               //start purging
               //-------------
               IF "APC".AUTOMATIC THEN 
                   IF ("APC".TI[0] <= REAL_TO_INT("PAR_MAIN".PD_PRG_TME)) AND NOT "PDI".FCH_APS  THEN 
                       //purging through V5
                       //------------------
                       IF (REAL_TO_INT("PAR_MAIN".PD_PRG_INLET_V5) = 1)   THEN 
                           "DC".V4_OP            :=  FALSE;
                           "DC".V5_OP            :=  TRUE;
                           "AC".SET_GAS_2_FLW    :=  "PAR_MAIN".PD_PRG_GAS_FLW;
                       //purging through V4
                       //------------------
                       ELSE
                           "DC".V4_OP            :=  TRUE;
                           "DC".V5_OP            :=  FALSE;
                           "AC".SET_GAS_2_FLW    :=  0.0;
                       END_IF;
                   //purging over
                   //------------
                   ELSE 
                       "DC".V4_OP            :=  FALSE;
                       "DC".V5_OP            :=  FALSE;
                       "AC".SET_GAS_2_FLW    :=  0.0;

                       #end_of_step[0] := true;                            

                   END_IF;
               END_IF;

               //calculate step time countdown
               //-----------------------------            
               "APC".ACT_TME_STE   := REAL_TO_INT("PAR_MAIN".PD_PRG_TME) - "APC".TI[0];

               #next_step[0] := 180;   

   //-step-180---level--0-------------------------------------------------------------                                                 
   //            PD: check if additional purge cycle is requested
   //---------------------------------------------------------------------------------                                                 
           180 :                                                     
               IF #next_step[0] = #active_step[0] THEN
                   "APC".OP_MSG  := "OP_MSG".BLANK;       
                   "APC".TI[0]   :=  0;            
                   #prg_cyc_cnt :=  #prg_cyc_cnt + 1;    //count amount of purge cycles                              
               END_IF;

               //delay switching to next step
               //----------------------------
               IF ("APC".TI[0] > 2) THEN
                   #end_of_step[0] := true;                            
               END_IF;

               //select next step
               //----------------
               IF (#prg_cyc_cnt >= REAL_TO_INT("PAR_MAIN".PD_AMT_PRG_CYC)) THEN
                   #next_step[0] := 200; 
               ELSE
                   #next_step[0] := 140; 
               END_IF;

   //-step-200---level--0-------------------------------------------------------------                                                 
   //            PD: pump down to 10 mbar
   //---------------------------------------------------------------------------------                                                 
           200 :                                                     
               IF #next_step[0] = #active_step[0] THEN                       
                   //reset initial temperature and power setpoints
                   //---------------------------------------------
                   "DIS".HTR_1_TMP_SET_PHA_STR   :=  0.0;
                   "DIS".HTR_2_PWR_SET_PHA_STR   :=  0.0;
                   "APC".TI[0]                   :=  0;                              // start pd time                              
                   "APC".OP_MSG                  :=  "OP_MSG".PD_10MBAR;
                   "APC".ACT_TME_STE             :=  0;
               END_IF;

               // calculate all setpoints 
               // -----------------------
               "AM_PAR_FNC_PD" (act_x_value := 0.0);

               //open vacuum valves
               //------------------
               "DC".P1_ON             := TRUE;   // main pump on
               "AC".SET_CTL_VALVE_POS := 100.0;  

               //monitor pump down time 
               //----------------------
               IF "APC".AUTOMATIC THEN 
                   IF "BM_VAC_DB".V2_ONDELAY_OVER THEN                                 // vacuum valve release
                       IF (INT_TO_REAL("APC".TI[0]) > "PAR_MAIN".PD_10_MBAR_TME) THEN    // pump down time limit exceeded?
                           "FLT".PD_TIME_10MBAR  := TRUE;
                           "APC".OP_MSG          := "OP_MSG".PD_CHECK_TIME;
                           #cont_enable[0]      := true;
                       END_IF;

                       //check end condition
                       //-------------------
                       IF ("AV".ACT_PRS_FCH < 10.0)  THEN         // p < 10 mbar ?
                           #end_of_step[0] := true;
                       END_IF; 

                   ELSE
                       "APC".TI[0]:= 0;      //keep timer on zero until vacuum valve release 
                   END_IF;
               ELSE
                   "APC".TI[0]:= 0;      //keep timer on zero until vacuum valve release 
               END_IF;

               #next_step[0] := 300; 

   //-step-300---level--0-------------------------------------------------------------                                                 
   //            PD: pump down to 1 mbar
   //---------------------------------------------------------------------------------                                                 
           300 :                                                  
               IF #next_step[0] = #active_step[0] THEN                       
                   "FLT".PD_TIME_10MBAR := FALSE;
                   "APC".OP_MSG := "OP_MSG".PD_1MBAR;
               END_IF;

               // calculate all setpoints 
               // -----------------------
               "AM_PAR_FNC_PD" (act_x_value := 0.0);

               IF (INT_TO_REAL("APC".TI[0]) > "PAR_MAIN".PD_1_MBAR_TME) THEN     // limit reached ?
                   "FLT".PD_TIME_1MBAR := TRUE;
                   "APC".OP_MSG := "OP_MSG".PD_CHECK_TIME;
                   #cont_enable[0] := true;
               END_IF;

               IF ("AV".ACT_PRS_FCH < 1.0) THEN                       // p < 1 mbar ?
                   #end_of_step[0] := true;                            
               END_IF;

               #next_step[0] := 400; 

   //-step-400---level--0-------------------------------------------------------------                                                 
   //            PD: pump down to 0.1 mbar
   //---------------------------------------------------------------------------------                                                 
           400 :                                                  
               IF #next_step[0] = #active_step[0] THEN
                   "FLT".PD_TIME_1MBAR := FALSE;
                   "APC".OP_MSG := "OP_MSG".PD_01MBAR;
               END_IF;

               // calculate all setpoints 
               // -----------------------
               "AM_PAR_FNC_PD" (act_x_value := 0.0);

               IF ( INT_TO_REAL("APC".TI[0]) > "PAR_MAIN".PD_01_MBAR_TME) THEN    // limit reached ?
                   "FLT".PD_TIME_01MBAR  := TRUE;
                   "APC".OP_MSG          := "OP_MSG".PD_CHECK_TIME;
                   #cont_enable[0]      := true;
               END_IF;

               IF ("AV".ACT_PRS_FCH < 0.1) THEN                       // p < 0.1 mbar ? 
                   #end_of_step[0] := true;                            
               END_IF;

               #next_step[0] := 500; 

   //-step-500---level--0-------------------------------------------------------------                                                 
   //            PD: pump down to 0.05 mbar
   //---------------------------------------------------------------------------------                                                 
           500 :                                                  
               IF #next_step[0] = #active_step[0] THEN
                   "FLT".PD_TIME_01MBAR := FALSE;
                   "APC".OP_MSG := "OP_MSG".PD_005MBAR;
               END_IF;

               // calculate all setpoints 
               // -----------------------
               "AM_PAR_FNC_PD" (act_x_value := 0.0);

               IF (INT_TO_REAL("APC".TI[0]) > "PAR_MAIN".PD_005_MBAR_TME) THEN   // limit reached ?
                   "FLT".PD_TIME_005MBAR := TRUE;
                   "APC".OP_MSG          := "OP_MSG".PD_CHECK_TIME;
                   #cont_enable[0]      := true;
               END_IF;

               IF ("AV".ACT_PRS_FCH < 0.05) THEN                      // p < 0.05 mbar ? 
                   #end_of_step[0] := true;                            
               END_IF;

               #next_step[0] := 600; 


   //-step-600---level--0-------------------------------------------------------------                                                 
   //            PD: pump down to final pressure
   //---------------------------------------------------------------------------------                                                 
           600 :                                                  
               IF #next_step[0] = #active_step[0] THEN
                   "FLT".PD_TIME_005MBAR := FALSE;
                   "APC".OP_MSG := "OP_MSG".PD_FINAL;
               END_IF;

               // calculate all setpoints 
               // -----------------------
               "AM_PAR_FNC_PD" (act_x_value := 0.0);

               //bypass filter activated
               //-----------------------
               IF (("CNF".ACT_DVC_CNF AND 2#1000_0000_0000_0000_0000_0000_0000_0000) = 2#1000_0000_0000_0000_0000_0000_0000_0000) THEN 

                   //close valve V3.4 to bypass filter when pressure below 5 mbar
                   //-----------------------------------------------------------
                   IF ("DIS".ACT_PRS_BYP_FIL < 5.0) THEN
                       "DC".V3_4_OP  := FALSE;
                   END_IF;

                   //set global release bit of V1.1
                   //------------------------------
                   IF NOT "PDO".V3_4 THEN
                       "DC".V1_1_REL := TRUE;
                   END_IF;

                   //check end condition
                   //-------------------
                   IF (("AV".ACT_PRS_FCH < "PAR_MAIN".PD_FINAL_PRS) AND "DC".V1_1_REL) THEN         // final presssure ?      
                       #end_of_step[0] := true;                            
                   END_IF;
               //no bypass filter
               //----------------
               ELSE
                   //check end condition
                   //-------------------
                   IF ("AV".ACT_PRS_FCH < "PAR_MAIN".PD_FINAL_PRS) THEN         // final presssure ?      
                       #end_of_step[0] := true;                            
                   END_IF;
               END_IF;

               #next_step[0] := 650; 

   //-step-650---level--0-------------------------------------------------------------                                                 
   //            PD: wait time after reaching final pressure before leak test
   //---------------------------------------------------------------------------------                                                 
           650 :                                                  
               IF #next_step[0] = #active_step[0] THEN
                   "APC".OP_MSG  := "OP_MSG".PD_WAIT_TME;
                   "APC".TI[0]   := 0;
               END_IF;

               // calculate all setpoints 
               // -----------------------
               "AM_PAR_FNC_PD" (act_x_value := 0.0);

               //remaining wait time
               //-------------------
               "APC".ACT_TME_STE   := REAL_TO_INT("PAR_MAIN".PD_WAIT_TME_FIN_PRS) - "APC".TI[0];

               //check end condition
               //-------------------
               IF ("APC".TI[0] >= (REAL_TO_INT("PAR_MAIN".PD_WAIT_TME_FIN_PRS))) THEN      
                   #end_of_step[0] := true;                            
               END_IF;

               #next_step[0] := 700; 

   //-step-700---level--0-------------------------------------------------------------                                                 
   //            PD: close vacuum valve
   //---------------------------------------------------------------------------------                                                 
           700 :                                                  
               IF #next_step[0] = #active_step[0] THEN                       
                   "APC".OP_MSG := "OP_MSG".PD_LEAK_TEST;
               END_IF;

               // calculate all setpoints 
               // -----------------------
               "AM_PAR_FNC_PD" (act_x_value := 0.0);

               "AC".SET_CTL_VALVE_POS := 0.0;                // close throttle valve
               "DC".V1_OPEN_REQ      := FALSE;               // only EKZ 2700
               "DC".V1_CLOSE_REQ     := TRUE;
               "DC".P3_ON            := FALSE;               // P3 off

               // check end condition
               //--------------------
               IF NOT "LT".V1_OPEN THEN  // closed ? 
                   #end_of_step[0] := true;                            
               END_IF;

               #next_step[0] := 800; 


   //-step-800---level--0-------------------------------------------------------------                                                 
   //            PD: do leak test
   //---------------------------------------------------------------------------------                                                 
           800 :                                                  
               IF #next_step[0] = #active_step[0] THEN                       
                   "APC".TI[0] := 0;                              // start time for leak test                              
                   #prs_leak_test_start := "AV".ACT_PRS_FCH;           // save start pressure  
               END_IF;

               //store pressure value before leak test is starting (CDP)
               //-------------------------------------------------------
               "DIS".ACT_FNC_PRS_BEF_LKT :=  #prs_leak_test_start;

               // calculate all setpoints 
               // -----------------------
               "AM_PAR_FNC_PD" (act_x_value := 0.0);

               // leakrate = (p2-p1)*V/t
               // ----------------------
               IF ("APC".TI[0] > 0) THEN 
                   //leak rate calculation with main and bypass filter
                   //-------------------------------------------------
                   IF (("CNF".ACT_DVC_CNF AND 2#1000_0000_0000_0000_0000_0000_0000_0000) = 2#1000_0000_0000_0000_0000_0000_0000_0000) THEN 
                       "AV".LRT_EKZ := ("AV".ACT_PRS_FCH - #prs_leak_test_start) * ("CNF".VOLUME_LEAK_TEST + "CNF".VOLUME_MAIN_FIL + "CNF".VOLUME_BYP_FIL) / INT_TO_REAL("APC".TI[0]);
                   //leak rate calculation only with main filter
                   //-------------------------------------------
                   ELSE
                       "AV".LRT_EKZ := ("AV".ACT_PRS_FCH - #prs_leak_test_start) * ("CNF".VOLUME_LEAK_TEST + "CNF".VOLUME_MAIN_FIL) / INT_TO_REAL("APC".TI[0]);
                   END_IF;
               END_IF;

               IF ("AV".LRT_EKZ < 0.0) THEN
                   "AV".LRT_EKZ := 0.0;
               END_IF;

               // show actual values
               // ------------------
               "DIS".ACT_LEAKR_FNC := "AV".LRT_EKZ;
               "APC".ACT_TME_STE   := REAL_TO_INT("PAR_MAIN".PD_LEAKTEST_TME) - "APC".TI[0];

               // check if leak test time is over
               //--------------------------------
               IF ("APC".TI[0] >= "PAR_MAIN".PD_LEAKTEST_TME) THEN   // time for leak test ? 
                   #end_of_step[0] := true;
               END_IF;
               #next_step[0] := 900; 


   //-step-900---level--0-------------------------------------------------------------                                                 
   //            PD: check for max. leak rate
   //---------------------------------------------------------------------------------                                                 
           900 :
               // calculate all setpoints 
               // -----------------------
               "AM_PAR_FNC_PD" (act_x_value := 0.0);

               IF ("AV".LRT_EKZ > "PAR_MAIN".PD_MAX_LEAKRATE) THEN   // max. leakrate ?                   
                   "FLT".PD_LEAKTEST := TRUE;
                   "APC".OP_MSG      := "OP_MSG".PD_CHECK_LEAK_RATE;

                   #cont_enable[0]  := true;                      // wait for continue
                   #next_step[0]    := 950; 
                   //repeat leak test
                   //----------------
                   IF "KYD".PD_NEW_LKT   THEN
                       #end_of_step[0] := true;     // next step  
                       #next_step[0] := 200;            //repeat leak test

                   END_IF;

               ELSE
                   "FLT".PD_LEAKTEST := FALSE;
                   #end_of_step[0]  := true;                      // next step                            
                   #next_step[0]    := 950; 

               END_IF;

   //-step-950--level--0-------------------------------------------------------------                                                 
   //            PD: switch vacuum pump on if next phase is melting
   //---------------------------------------------------------------------------------    

           950 :             
               IF #next_step[0] = #active_step[0] THEN                       
                   "APC".TI[0]   := 0;                           // start wait time pump  
                   "APC".OP_MSG  := "OP_MSG".BLANK;                                          
               END_IF;

               IF ("APC".PD_WITH_ME) THEN                        // with melting ?
                   "DC".P1_ON := TRUE;
                   IF "BM_VAC_DB".V2_ONDELAY_OVER THEN           // wait until V2 delay is over
                       #end_of_step[0] := true;
                   END_IF;
               ELSE                                              
                   #end_of_step[0] := true;                     // switch to next step
               END_IF;

               #next_step[0] := 1000;



   //-step-1000--level--0-------------------------------------------------------------                                                 
   //            PD: start melting or switch to idle
   //---------------------------------------------------------------------------------                                                 
           1000 :                                                  

               "APC".ACT_TME_STE := 0;
               "FLT".PD_LEAKTEST := FALSE;

               IF ("APC".PD_WITH_ME) THEN                         // with melting ?
                   "DC".MOD_ME := TRUE;                           // switch to melting
               ELSE;
                  //DC.P1_ON := FALSE;                           // stop main pump 

                   // stop drives and reset setpoint values after leaktest with drives active
                   // -----------------------------------------------------------------------
                   IF "CNF".CONF_DRV_WHILE_LRT = TRUE THEN
                       "DC".XT_LFT_UP    := FALSE;                    // stop crystal lift
                       "DC".XT_LFT_DN    := FALSE;
                       "DC".XT_LFT_FST   := FALSE;
                       "DC".XT_ROT_CW    := FALSE;                    // stop crystal rotation
                       "DC".XT_ROT_CCW   := FALSE;

                       "DC".CR_LFT_UP    := FALSE;                    // stop crucible lift
                       "DC".CR_LFT_DN    := FALSE;
                       "DC".CR_LFT_FST   := FALSE;
                       "DC".CR_ROT_CW    := FALSE;                    // stop crucible rotation
                       "DC".CR_ROT_CCW   := FALSE;

                       "AC".SET_XT_SPD := 0.0;
                       "AC".SET_XT_ROT := 0.0;
                       "AC".SET_CR_SPD := 0.0;
                       "AC".SET_CR_ROT := 0.0;
                   END_IF;

                   "DC".MOD_ID := TRUE;                           // switch to idle 
               END_IF;

               #next_step[0] := 1000;                            // E N D

   //---------------------------------------------------------------------------------                                                 
   //---------------------------------------------------------------------------------                                                 

   //-error------level--0---------------------------------------------------(error in level 0)-------------
       ELSE:                                                        
           //error code                                                //do error code
           ;        
   //------------------------------------------------------------------------------------------------------
       END_CASE;

       #start_previous := #start;                                    //save start input for next call 
       #cont_previous := "APC".CONT;                                  //save cont input for next call 
       #resume_previous := "APC".RESUME;                              //save resume input for next call
       #jump_previous := "APC".JUMP;                                  //save jump input for next call
       #single_previous := "APC".SINGLE;                              //save single input for next call
END_FUNCTION_BLOCK

FUNCTION_BLOCK "AM_ME"   // FB197, SCL
{ S7_Optimized_Access := 'FALSE' }
VERSION : 0.0
// --------------------------------------------------------------------------------
//     program     :    AM_ME
//     description :    apc melting module  
//     name        :    D. Bruess
//     date        :    04.11.99
// 
//     revision    :    change default rotation direction: xtal= ccw and cruc= cw
//     name        :    G. Eibelsh鋟ser
//     date        :    26.04.00
//     
//                     (c)CGS
//     --------------------------------------------------------------------------------
   VAR_INPUT
      start : Bool;   // start sequence, activate step 10 (impulse triggered)
   END_VAR
   VAR
      start_previous : Bool;   // start input value of last call
      cont_previous : Bool;   // cont input value of last call
      resume_previous : Bool;   // resume input value of last call
      jump_previous : Bool;   // jump input value of last call
      single_previous : Bool;   // single input value of last call
      active_step : Array[0..7] of Int;   // active step number for sequence level 0..7
      next_step : Array[0..7] of Int;   // next step number for sequence level 0..7
      hold_step : Array[0..7] of Int;   // step number of step on hold
      end_of_step : Array[0..7] of Bool;   // active step is done flag for sequence 0..7
      EndOfStep : Bool;   // default value for active step is done flag
      cont_enable : Array[0..7] of Bool;   // enable continue function
      ContEnable : Bool;   // default value for enable continue function
      cam_active : Bool;   // camera used for this step
      cruc_in_pos : Bool;   // crucible in new position
      next_step_fdr : Bool;
      check_mlt_lvl_done : Bool;
      step_switch_done : Bool;
      next_melt_step : Bool;
      act_step_fdr : Int;
      par_line : Int;   // act. line from parameter table
      par_step : Int;   // number of this step
      par_time : Int;   // time parameter for this step
      set_cr_pos_old : Real;   // old setpoint for crucible position
      htr_1_pwr_act_step : Real;
      htr_1_pwr_next_step : Real;
   END_VAR
   VAR CONSTANT
      max_amt_of_steps : Int := 21;   // maximum amount of step lines
   END_VAR
BEGIN

       "APC".STATUS := "APC".MELTING;                                  // set apc status               

       "AM_SEQUENCE_CTL" (start_p            := #start,               // control sequence
                        start_previous_p   := #start_previous,
                        cont_previous_p    := #cont_previous, 
                        resume_previous_p  := #resume_previous,
                        jump_previous_p    := #jump_previous,
                        single_previous_p  := #single_previous,
                        active_step_p      := #active_step, 
                        next_step_p        := #next_step,
                        hold_step_p        := #hold_step, 
                        end_of_step_p      := #end_of_step, 
                        cont_enable_p      := #cont_enable); 

       //Set the "Oxidation valve" in all Phases
       "DC".V21_OP:= DINT_TO_BOOL(REAL_TO_DINT("PAR_MAIN".ME_V21_OPEN));

       CASE #active_step[0] OF    //sequence level_0
       //step--0-----level--0-------------------------------------------------off--(sequence off)--------------
           0    :                                                  
                #next_step[0] := 0;

       //step--1-----level--0-------------------------------------------------hold-(test sequence)-------------
           1   :                                                       
               IF #next_step[0] = #active_step[0] THEN                   //init step     
                   //init code
                   ; 
               END_IF;

               //step code                                             //do step
               ;

       //-step-10----level--0----------------------------------------------main-(start sequence)---------------                                                 

       //-step-10----level--0-------------------------------------------------------------                                                 
       //            ME: init melting sequence
       //---------------------------------------------------------------------------------                                                 
           10  :                                                     

               // init vacuum system
               // ------------------
               "DC".V3_OP    := FALSE;
               "DC".V4_OP    := FALSE;
               "DC".V5_OP    := TRUE;                         // open V5
               "DC".V6_OP    := FALSE;
               "DC".V8_OP    := FALSE;
               "DC".V11_OP   := FALSE;
               "DC".V11_CL   := TRUE;
               "DC".V12_OP   := FALSE;
               "DC".V13_OP   := FALSE;
               "DC".V20_OP   := FALSE;
               "DC".V22_OP   := FALSE;
               "DC".V24_OP   := FALSE;
               "DC".P1_ON    := TRUE;                         // start main pump
               "DC".P3_ON    := FALSE;
               "DC".V3_4_OP  := FALSE;
               "DC".V1_1_REL := FALSE;

               "DC".V3_2_OP := FALSE;

               "DC".V1_OPEN_REQ   := FALSE;                // only EKZ 2700
               "DC".V1_CLOSE_REQ  := FALSE;

               // init drives
               // -----------
               "DC".XT_LFT_UP    := FALSE;                    // stop crystal lift
               "DC".XT_LFT_DN    := FALSE;
               "DC".XT_LFT_FST   := FALSE;
               "DC".XT_ROT_CW    :=      "BM_ROT_DRV_DIR_DB".ROT_DIR   AND ("AC".SET_XT_ROT <> 0.0);
               "DC".XT_ROT_CCW   := NOT  "BM_ROT_DRV_DIR_DB".ROT_DIR   AND ("AC".SET_XT_ROT <> 0.0);

               "DC".CR_LFT_UP    := FALSE;                    // stop crucible lift
               "DC".CR_LFT_DN    := FALSE;
               "DC".CR_LFT_FST   := FALSE;
               "DC".CR_ROT_CW    := NOT  "BM_ROT_DRV_DIR_DB".ROT_DIR   AND ("AC".SET_CR_ROT <> 0.0);
               "DC".CR_ROT_CCW   :=      "BM_ROT_DRV_DIR_DB".ROT_DIR   AND ("AC".SET_CR_ROT <> 0.0);

               "AC".SET_XT_SPD := 0.0;
               "AC".SET_XT_ROT := "KYA".SET_XT_ROT;
               "AC".SET_CR_SPD := 0.0;
               "AC".SET_CR_ROT := "KYA".SET_CR_ROT;

               #set_cr_pos_old := -1.0;

               // init heater
               // -----------
               "DC".HTR_1_ON := ("AC".SET_HTR_1_PWR > 0.0);
               "DC".HTR_2_ON := ("AC".SET_HTR_2_PWR > 0.0);
               "DC".HTR_3_ON := FALSE;

               "AC".SET_HTR_1_PWR := "KYA".SET_HTR_1_PWR;
               "AC".SET_HTR_2_PWR := "KYA".SET_HTR_2_PWR;
               "AC".SET_HTR_3_PWR := 0.0;

               //mobile feeder
               //-------------
               "DC".MOB_FDR_MVE_IN_SEQ_ON    :=  FALSE;
               IF ("LT".MOB_FDR_DCK_DONE AND ("DV".FDG_MVE_IN_SEQ_DONE OR NOT "DV".FDG_MVE_OUT_SEQ_DONE)) THEN 
                   "DC".MOB_FDR_MVE_OUT_SEQ_ON   :=  TRUE;
               ELSE
                   "DC".MOB_FDR_MVE_OUT_SEQ_ON   :=  FALSE;
               END_IF;
               "DC".MOB_FDR_VIB_ON           :=  FALSE;
               "FLT".MOB_FDR_NOT_DCK         :=  FALSE;
               "FLT".MOB_FDR_STP_PARA        :=  FALSE;

               // init magnet
               // -----------
               "DC".MAG_ON := ("AC".SET_MAG_1_CUR > 0.0);                       

               "AC".SET_MAG_1_CUR := "KYA".SET_MAG_1_CUR;
               "AC".SET_MAG_2_CUR := "KYA".SET_MAG_1_CUR * "KYA".SET_MAG_RATIO_CUR;

               // init control loops
               // ------------------
               "DC".CTL_DIA_ON := FALSE;                   // all control loops off
               "DC".CTL_GRW_RTE_ON := FALSE;
               "DC".CTL_PULL_RTE_ON := FALSE;
               "DC".CTL_CRUC_ROT_ON := FALSE;
               "DC".CTL_MLT_LVL_ON := FALSE;
               "DC".CTL_MLT_1_TMP_ON := FALSE;
               "DC".CTL_MLT_2_TMP_ON := FALSE;
               "DC".CTL_MLT_DRIFT_ON := FALSE;
               "DC".CTL_GAP_ON       := FALSE;
               "DC".CTL_HTR_1_TMP_ON := FALSE;
             //DC.CTL_HTR_2_TMP_ON := FALSE;
               "DC".SET_HTR_1_TMP_ABS := TRUE;             // disable inc functions
               "DC".SET_HTR_2_PWR_ABS := TRUE;

               "DC".CTL_PRS_ON := TRUE;                    // pressure control on

               "DC".CTL_SI_FDR_ON := FALSE;
               "DC".CTL_DOP_FDR_ON := FALSE;

               "AC".SET_XT_DIA := 0.0;
               "AC".SET_GRW_RTE := 0.0;
               "AC".SET_AVG_SPD := 0.0;
               "AC".SET_AVG_CRUC_ROT := 0.0;
               "AC".SET_MLT_LVL_LSR := 0.0;
               "AC".SET_MLT_1_TMP := 0.0;
               "AC".SET_MLT_2_TMP := 0.0;
               "AC".SET_HTR_1_TMP := 0.0;
               "AC".SET_HTR_2_TMP := 0.0;

               // init measurement system
               // -----------------------
               "DC".CAM_ISP_ON   :=  TRUE;      //inspection off
               "DC".CAM_INIT     :=  FALSE;
               "DC".CAM_MLT      :=  TRUE;
               "DC".CAM_DIP      :=  FALSE;
               "DC".CAM_DIA      :=  FALSE;            
               "DC".CAM_SEL_1    :=  TRUE;
               "DC".CAM_SEL_2    :=  FALSE;

               "KYA".SET_THR_CAL_FACT    := 1.0;           // default value for threshold ratio factor
               "DV".THR_CALC_DISABLED    := TRUE;

               "DC".LSR_ON       := FALSE;                 // laser off
               "DV".MLT_LVL_FND  := FALSE;                
               "DC".MCC_ON       := FALSE;                 // melt contact control off
               "DC".MCC_TST_ON   := FALSE;

               // init Si feeder system
               // ---------------------
               "DC".SI_FDR_ON := FALSE;                    // feeder off
               "DC".DOP_FDR_ON := FALSE;

               "AC".SET_FDR_SI := 0.0;
               "AC".SET_FDR_DOP := 0.0;
               #act_step_fdr := 10;

               // init lamp on control cabinet
               // ----------------------------
               "DV".LMP_OR := false;

               // calculate all setpoints (step no. from 1st line of seqence table)
               // ----------------------------------------------------------------
               #par_line := 1;
               #par_step := REAL_TO_INT ("PAR_X_VALUES_1".PAR["APC".MELTING, #par_line]);            
               "AM_PAR_FNC_ME" (act_x_value := #par_step);


               // process control flags
               // ---------------------
               "APC".PNBDY := FALSE;
               "APC".BYRST := FALSE;


               // enable automatic mode
               // ---------------------
               "DC".MOD_AUT_ENB := TRUE;

               #end_of_step[0] := true;                            
               #next_step[0] := 100;


       //-step-100---level--0-------------------------------------------------------------                                                 
       //            ME: wait for automatic mode
       //---------------------------------------------------------------------------------                                                 
           100 :                                                     
               IF #next_step[0] = #active_step[0] THEN
                   "APC".OP_MSG := "OP_MSG".WAIT_FOR_AUTO;                                                  
               END_IF;

               IF "APC".AUTOMATIC = TRUE THEN                     // automatic mode ?
                   #end_of_step[0] := true;                            
               END_IF;                                    
               #next_step[0] := 150;


       //-step-150---level--0-------------------------------------------------------------                                                 
       //            ME: start melting time
       //---------------------------------------------------------------------------------                                                 
           150 :                                                     
               "APC".ACT_TME_PROC := 0;                           // start process time
               #end_of_step[0] := true;                            
               #next_step[0] := 200;


       //-step-200---level--0-------------------------------------------------------------                                                 
       //            ME: do one melting step
       //---------------------------------------------------------------------------------                                                 
           200 :                                                     
               IF #next_step[0] = #active_step[0] THEN                     
                   //reset initial temperature and power setpoints
                   //---------------------------------------------
                   "DIS".HTR_1_TMP_SET_PHA_STR   :=  0.0;
                   "DIS".HTR_2_PWR_SET_PHA_STR   :=  0.0;

                   "APC".TI[0]                   :=  0;          // start step time
                   "APC".TI[1]                   :=  0;

               END_IF;

               // fetch actual step number and time for this step
               // -----------------------------------------------
               #par_step := REAL_TO_INT ("PAR_X_VALUES_1".PAR["APC".MELTING, #par_line]);            
               #par_time := REAL_TO_INT ("PAR_TME".PAR["APC".MELTING, #par_line]);

               // set flag for active camera step
               // -------------------------------
               #cam_active  := ("PAR_MAIN".ME_DETECT_STEP = #par_step);

               //set melt check flag
               //-------------------
               "DV".CAM_MLT_CHK  :=  #cam_active;

               // show actual step number
               // -----------------------
               "APC".OP_MSG := #par_step;

               // calculate all setpoints for this step
               // -------------------------------------                                      
               "AM_PAR_FNC_ME" (act_x_value := #par_step);

               // call drive module for crucible positioning
               // ------------------------------------------
               IF ("AV".SET_CR_POS <> #set_cr_pos_old) THEN
                 #cruc_in_pos := FALSE;
               END_IF;

               "DC".CR_LFT_FST := TRUE;

               "AM_CR_DRV_MOVE_DB"  (set_pos := "AV".SET_CR_POS,
                                               set_spd := "AV".SET_CR_SPD,
                                               act_pos := "AV".ACT_CR_POS,
                                               cnf     := "CNF".CNF_CR_POS,
                                               out_up  := "DC".CR_LFT_UP,
                                               out_dn  := "DC".CR_LFT_DN,
                                               out_spd := "AC".SET_CR_SPD,
                                               done    := #cruc_in_pos);

               IF (#cruc_in_pos) THEN
                 #set_cr_pos_old := "AV".SET_CR_POS;
               END_IF;

               // control heater
               // --------------
               "DC".HTR_1_ON := ("AC".SET_HTR_1_PWR > 0.0);
               "DC".HTR_2_ON := ("AC".SET_HTR_2_PWR > 0.0);

               //mobile feeder 
               //-------------
               IF (REAL_TO_INT("PAR_MAIN".ME_FDR_STEP) > 0) THEN  
                   //verify feeder step parameters
                   //-----------------------------
                   IF (((REAL_TO_INT("PAR_MAIN".ME_FDR_STEP + "PAR_MAIN".ME_AMT_OF_FDG_STP)) > 21) OR (REAL_TO_INT("PAR_MAIN".ME_AMT_OF_FDG_STP) = 0)) THEN
                       "FLT".MOB_FDR_STP_PARA    :=  TRUE;
                   ELSE
                       "FLT".MOB_FDR_STP_PARA    :=  FALSE;
                   END_IF;

                   //feeder is docked to puller
                   //--------------------------
                   IF "LT".MOB_FDR_DCK_DONE THEN 
                       //activation of feeder move in sequence
                       //-------------------------------------
                       IF ((#par_step >= REAL_TO_INT("PAR_MAIN".ME_FDR_STEP)) AND NOT "DC".MOB_FDR_MVE_OUT_SEQ_ON) THEN 
                           "DC".MOB_FDR_MVE_IN_SEQ_ON    :=  TRUE;
                           "FLT".MOB_FDR_NOT_DCK         :=  FALSE;
                       END_IF;

                       //activation of feeder move out sequence
                       //--------------------------------------
                       IF ((#par_step >= REAL_TO_INT("PAR_MAIN".ME_FDR_STEP + "PAR_MAIN".ME_AMT_OF_FDG_STP)) AND NOT "FLT".MOB_FDR_STP_PARA) THEN 
                           "DC".MOB_FDR_MVE_OUT_SEQ_ON   :=  TRUE;
                           "DC".MOB_FDR_MVE_IN_SEQ_ON    :=  FALSE;
                       ELSE
                           "DC".MOB_FDR_MVE_OUT_SEQ_ON   :=  FALSE;
                       END_IF;

                       //activation of feeder vibration after drive in sequence is done
                       //--------------------------------------------------------------
                       IF ("DV".FDG_MVE_IN_SEQ_DONE AND NOT "DC".MOB_FDR_MVE_OUT_SEQ_ON) THEN
                           "DC".MOB_FDR_VIB_ON   :=  ("AC".SET_MOB_FDR_VIB_FRQ >= 0.1);
                       ELSE
                           "DC".MOB_FDR_VIB_ON   :=  FALSE;
                       END_IF;

                   //set alarm when feeder is not docked in requested feeding step
                   //-------------------------------------------------------------    
                   ELSIF (#par_step = REAL_TO_INT("PAR_MAIN".ME_FDR_STEP)) THEN 
                       "FLT".MOB_FDR_NOT_DCK :=  TRUE;
                   END_IF;
               ELSE
                   "DC".MOB_FDR_MVE_IN_SEQ_ON    :=  FALSE;
                   "DC".MOB_FDR_VIB_ON           :=  FALSE;
               END_IF;

               // control magnet
               // --------------
               "DC".MAG_ON := ("AC".SET_MAG_1_CUR > 0.0);

               "AC".SET_MAG_1_CUR := "AV".SET_MAG_1_CUR;
               "AC".SET_MAG_2_CUR := "AV".SET_MAG_1_CUR * "AV".SET_MAG_RATIO_CUR;

               // control rotation
               // ----------------
               "DC".XT_ROT_CW    :=      "BM_ROT_DRV_DIR_DB".ROT_DIR   AND ("AC".SET_XT_ROT <> 0.0);
               "DC".XT_ROT_CCW   := NOT  "BM_ROT_DRV_DIR_DB".ROT_DIR   AND ("AC".SET_XT_ROT <> 0.0);

               "DC".CR_ROT_CW    := NOT  "BM_ROT_DRV_DIR_DB".ROT_DIR   AND ("AC".SET_CR_ROT <> 0.0);
               "DC".CR_ROT_CCW   :=      "BM_ROT_DRV_DIR_DB".ROT_DIR   AND ("AC".SET_CR_ROT <> 0.0);

               // time till end of this step
               // --------------------------
               "APC".ACT_TME_STE := #par_time - "APC".TI[0];

               // end of step ?
               // -------------
               IF        (("APC".TI[0] > #par_time)                                                   //step time over
                   AND     #cruc_in_pos                                                             //crucible in positon
                   AND   ((#cam_active AND "DV".CAM_MELT_COMPLETE)  OR NOT #cam_active))         THEN  //melt complete

                   #end_of_step[0] := true;

               END_IF;

               #next_step[0] := 300; 

       //-step-300---level--0-------------------------------------------------------------                                                 
       //            ME: transition to next step, check for last step
       //---------------------------------------------------------------------------------                                                 
           300 :                                                  
               IF #next_step[0] = #active_step[0] THEN                       
                   // next line in parameter table
                   // ----------------------------
                   #par_line := #par_line + 1;
               END_IF;

               // fetch step number of this new line
               // ----------------------------------
               IF (#par_line <= 21) THEN
                   #par_step := REAL_TO_INT ("PAR_X_VALUES_1".PAR["APC".MELTING, #par_line]);            
               END_IF;


               // step number = 0 or last line ? 
               // ------------------------------
               IF ((#par_step = 0)
                   OR (#par_line > 21) ) THEN

                   // start dipping
                   // -------------
                   #end_of_step[0] := true;                            
                   #next_step[0] := 400; 
               ELSE
                   // continue with next melting step
                   // -------------------------------
                   #end_of_step[0] := true;                            
                   #next_step[0] := 200; 
               END_IF;

       //-step-400---level--0-------------------------------------------------------------                                                 
       //            ME: start dipping mode
       //---------------------------------------------------------------------------------                                                 
           400 :                                                  
               IF #next_step[0] = #active_step[0] THEN
                   "APC".OP_MSG := "OP_MSG".BLANK;
               END_IF;

               //select next phase according selected machine state
               //--------------------------------------------------
               IF ("STA".ACT_STATE = "APC".STATE_BAKE_OUT) THEN        //state bake out is selected
                   "DC".MOD_SD   := TRUE;                            //switch to shut down
               ELSE
                   "DC".MOD_DI   := TRUE;                            //switch to dipping
               END_IF;

               #next_step[0]        := 400;                 //E N D 

       //---------------------------------------------------------------------------------                                                 
       //-error------level--0---------------------------------------------------(error in level 0)-------------
       ELSE:                                                        
           //error code                                                //do error code
           ;        
   //------------------------------------------------------------------------------------------------------
       END_CASE;

       CASE #active_step[1] OF    //sequence level_1
   //step--0-----level--1-------------------------------------------------off--(sequence off)--------------
           0    :                                                  
                #next_step[1] := 0;

   //step--1-----level--1-------------------------------------------------hold-(test sequence)-------------
           1   :                                                       
               IF #next_step[1] = #active_step[1] THEN                   //init step     
                   //init code
                   ; 
               END_IF;

               //step code                                             //do step
               ;

   //-step-10----level--1----------------------------------------------main-(start sequence)---------------                                                 
           10  :                                                     
               IF #next_step[1] = #active_step[1] THEN                   //init step     
                   //init code 
                   ;                                                  
               END_IF;

               //step code                                             //do step
               ;
               IF #ContEnable = true THEN                               //enable continue function
                   #cont_enable[1] := true;
               END_IF;
               IF #EndOfStep = true THEN                                //define end of step condition
                   #end_of_step[1] := true;                            
               END_IF;                                    
               #next_step[1] := 0;                                      //define next step #
               IF #end_of_step[1] = true THEN                           //do on transition
                   //transition code
                   ;
               END_IF;

   //-step-100---level--1----------------------------------------------name-(remarks)----------------------                                                 
           100 :                                                     
               IF #next_step[1] = #active_step[1] THEN                   //init step     
                   //init code 
                   ;                                                  
               END_IF;

               //step code                                             //do step
               ;
               IF #ContEnable = true THEN                               //enable continue function
                   #cont_enable[1] := true;
               END_IF;
               IF #EndOfStep = true THEN                                //define end of step condition
                   #end_of_step[1] := true;                            
               END_IF;                                    
               #next_step[1] := 0;                                      //define next step #
               IF #end_of_step[1] = true THEN                           //do on transition
                   //transition code
                   ;
               END_IF;

   //-step-200---level--1----------------------------------------------name-(remarks)----------------------                                                 
           200 :                                                     
               IF #next_step[1] = #active_step[1] THEN                   //init step     
                   //init code 
                   ;                                                  
               END_IF;

               //step code                                             //do step
               ;
               IF #ContEnable = true THEN                               //enable continue function
                   #cont_enable[1] := true;
               END_IF;
               IF #EndOfStep = true THEN                                //define end of step condition
                   #end_of_step[1] := true;                            
               END_IF;                                    
               #next_step[1] := 0;                                      //define next step #
               IF #end_of_step[1] = true THEN                           //do on transition
                   //transition code
                   ;
               END_IF;

   //-error------level--1---------------------------------------------------(error in level 1)-------------
       ELSE:                                                        
           //error code                                                //do error code
           ;        
   //------------------------------------------------------------------------------------------------------
   END_CASE;

   CASE #active_step[2] OF    //sequence level_2
   //step--0-----level--2-------------------------------------------------off--(sequence off)--------------
           0    :                                                  
                #next_step[2] := 0;

   //step--1-----level--2-------------------------------------------------hold-(test sequence)-------------
           1   :                                                       
               IF #next_step[2] = #active_step[2] THEN                   //init step     
                   //init code
                   ; 
               END_IF;

               //step code                                             //do step
               ;

   //-step-10----level--2----------------------------------------------main-(start sequence)---------------                                                 
           10  :                                                     
               IF #next_step[2] = #active_step[2] THEN                   //init step     
                   //init code 
                   ;                                                  
               END_IF;

               //step code                                             //do step
               ;
               IF #ContEnable = true THEN                               //enable continue function
                   #cont_enable[2] := true;
               END_IF;
               IF #EndOfStep = true THEN                                //define end of step condition
                   #end_of_step[2] := true;                            
               END_IF;                                    
               #next_step[1] := 0;                                      //define next step #
               IF #end_of_step[2] = true THEN                           //do on transition
                   //transition code
                   ;
               END_IF;

   //-step-100---level--2----------------------------------------------name-(remarks)----------------------                                                 
           100 :                                                     
               IF #next_step[2] = #active_step[2] THEN                   //init step     
                   //init code 
                   ;                                                  
               END_IF;

               //step code                                             //do step
               ;
               IF #ContEnable = true THEN                               //enable continue function
                   #cont_enable[2] := true;
               END_IF;
               IF #EndOfStep = true THEN                                //define end of step condition
                   #end_of_step[2] := true;                            
               END_IF;                                    
               #next_step[2] := 0;                                      //define next step #
               IF #end_of_step[2] = true THEN                           //do on transition
                   //transition code
                   ;
               END_IF;

   //-error------level--2---------------------------------------------------(error in level 2)-------------
       ELSE:                                                        
           //error code                                                //do error code
           ;        
   //------------------------------------------------------------------------------------------------------
       END_CASE;

       #start_previous := #start;                                    //save start input for next call 
       #cont_previous := "APC".CONT;                                  //save cont input for next call 
       #resume_previous := "APC".RESUME;                              //save resume input for next call
       #jump_previous := "APC".JUMP;                                  //save jump input for next call
       #single_previous := "APC".SINGLE;                              //save single input for next call
END_FUNCTION_BLOCK

FUNCTION_BLOCK "AM_DI"   // FB198, SCL
{ S7_Optimized_Access := 'FALSE' }
VERSION : 0.0
// --------------------------------------------------------------------------------
//     program     :    AM_DI
//     description :    apc dipping module  
//     name        :    G. Eibelsh鋟ser
//     date        :    31.01.00
// 
//     revision    :    call AM_SEQUENCE_CTL
//     name        :    D. Bruess
//     date        :    26.10.99
//     
//     revision    :    change default rotation direction: xtal= ccw and cruc= cw
//     name        :    G. Eibelsh鋟ser
//     date        :    26.04.00
// 
// 
//                     (c)CGS
//     --------------------------------------------------------------------------------
   VAR_INPUT
      start : Bool;   // start sequence, activate step 10 (impulse triggered)
   END_VAR
   VAR
      start_previous : Bool;   // start input value of last call
      cont_previous : Bool;   // cont input value of last call
      resume_previous : Bool;   // resume input value of last call
      jump_previous : Bool;   // jump input value of last call
      single_previous : Bool;   // single input value of last call
      active_step : Array[0..7] of Int;   // active step number for sequence level 0..7
      next_step : Array[0..7] of Int;   // next step number for sequence level 0..7
      hold_step : Array[0..7] of Int;   // step number of step on hold
      end_of_step : Array[0..7] of Bool;   // active step is done flag for sequence 0..7
      cont_enable : Array[0..7] of Bool;   // enable continue function
      EndOfStep : Bool;   // default value for active step is done flag
      ContEnable : Bool;   // default value for enable continue function
      par_line : Int;   // act. line from parameter table
      par_step : Int;   // number of this step
      par_time : Int;   // time parameter for this step
      htr_1_tmp_before_gap : Real;   // save heater 1 temperature before gap
      cruc_in_pos : Bool;   // crucible in position for stabilisation
      xtal_in_pos : Bool;   // xtal in position for stabilisation
      dip_temp_dev_ok : Bool;   // dip temp deviation within the temp band
      thr_adj_ok : Bool;   // threshold adjustment done or disabled
      dip_condition_ok : Bool;   // dip conditions are ok
      mcc_error_flag_1 : Bool;   // mcc_enable = on, mcc_test = on
      mcc_error_flag_2 : Bool;   // mcc_enable = off, mcc_test = off
      mcc_isolation_flag : Bool;   // mcc_enable = on, mcc_test = off
      xt_lgh_calc_done : Bool;   // calculation of 2nd crystal length done
      xt_wgt_chgd : Bool;   // crystal weight of grown crystal was changed
      set_cr_pos_old : Real;   // old position setpoint for cruc.
      ne_mlt_con_pos : Real;   // melt contact position of previous neck
      prv_calc_wgt_grw_xt : Real;   // previous calculated value of last crystal weight
      di_neck_rmlt_len : Real;   // remelt length of previous neck
   END_VAR
   VAR_TEMP
      dip_image_check : Bool;   // status for dip image verification
   END_VAR
BEGIN

       "APC".STATUS := "APC".DIPPING;                                  // set apc status               

       "AM_SEQUENCE_CTL" (start_p            := #start,               // control sequence
                        start_previous_p   := #start_previous,
                        cont_previous_p    := #cont_previous, 
                        resume_previous_p  := #resume_previous,
                        jump_previous_p    := #jump_previous,
                        single_previous_p  := #single_previous,
                        active_step_p      := #active_step, 
                        next_step_p        := #next_step,
                        hold_step_p        := #hold_step, 
                        end_of_step_p      := #end_of_step, 
                        cont_enable_p      := #cont_enable); 

       //Set the "Oxidation valve" in all Phases
       "DC".V21_OP:= DINT_TO_BOOL(REAL_TO_DINT("PAR_MAIN".DI_V21_OPEN));

       CASE #active_step[0] OF    //sequence level_0
   //step--0-----level--0-------------------------------------------------off--(sequence off)--------------
           0    :                                                  
                #next_step[0] := 0;

   //step--1-----level--0-------------------------------------------------hold-(test sequence)-------------
           1   :                                                       
               IF #next_step[0] = #active_step[0] THEN                   //init step     
                   //init code
                   ; 
               END_IF;

               //step code                                             //do step
               ;

   //-step-10----level--0----------------------------------------------main-(start sequence)---------------                                                 

   //-step-10----level--0-------------------------------------------------------------                                                 
   //            DI: init dipping sequence
   //---------------------------------------------------------------------------------                                                 
           10  :                                                     

               // init vacuum system
               // ------------------
               "DC".V1_OP    := TRUE;
               "DC".V3_OP    := FALSE;
               "DC".V4_OP    := FALSE;
               "DC".V5_OP    := TRUE;
               "DC".V6_OP    := FALSE;
               "DC".V8_OP    := FALSE;
               "DC".V11_OP   := FALSE;
               "DC".V11_CL   := TRUE;
               "DC".V12_OP   := FALSE;
               "DC".V13_OP   := FALSE;
               "DC".V20_OP   := FALSE;
               "DC".V22_OP   := FALSE;
               "DC".V24_OP   := FALSE;
               "DC".P1_ON    := TRUE;                         // start main pump
               "DC".P3_ON    := FALSE;
               "DC".V3_4_OP  := FALSE;
               "DC".V1_1_REL := FALSE;

               "DC".V3_2_OP  := FALSE;                      // vacuum valve feeder

               "DC".V1_OPEN_REQ   := FALSE;                // only EKZ 2700
               "DC".V1_CLOSE_REQ  := FALSE;

               // init drives
               // -----------
               "DC".XT_LFT_UP := FALSE;                    // stop crystal lift
               "DC".XT_LFT_DN := FALSE;
               "DC".XT_LFT_FST := FALSE;
               "DC".XT_ROT_CW := "BM_ROT_DRV_DIR_DB".ROT_DIR;            //1 = cw
               "DC".XT_ROT_CCW := NOT "BM_ROT_DRV_DIR_DB".ROT_DIR;       //0 = ccw

               "DC".CR_LFT_UP := FALSE;                    // stop crucible lift
               "DC".CR_LFT_DN := FALSE;
               "DC".CR_LFT_FST := FALSE;
               "DC".CR_ROT_CW := NOT "BM_ROT_DRV_DIR_DB".ROT_DIR;        //0 = cw
               "DC".CR_ROT_CCW := "BM_ROT_DRV_DIR_DB".ROT_DIR;           //1 = ccw

               "AC".SET_XT_SPD := 0.0;
               "AC".SET_XT_ROT := "KYA".SET_XT_ROT;
               "AC".SET_CR_SPD := 0.0;
               "AC".SET_CR_ROT := "KYA".SET_CR_ROT;

               #set_cr_pos_old := -1.0;

               // init heater
               // -----------
               "DC".HTR_1_ON := TRUE;                      // heater on
               "DC".HTR_2_ON := TRUE;
               "DC".HTR_3_ON := FALSE;

               "AC".SET_HTR_1_PWR := "KYA".SET_HTR_1_PWR;
               "AC".SET_HTR_2_PWR := "KYA".SET_HTR_2_PWR;
               "AC".SET_HTR_3_PWR := 0.0;

               //mobile feeder
               //-------------
               "DC".MOB_FDR_MVE_IN_SEQ_ON    :=  FALSE;
               IF ("LT".MOB_FDR_DCK_DONE AND ("DV".FDG_MVE_IN_SEQ_DONE OR NOT "DV".FDG_MVE_OUT_SEQ_DONE)) THEN 
                   "DC".MOB_FDR_MVE_OUT_SEQ_ON   :=  TRUE;
               ELSE
                   "DC".MOB_FDR_MVE_OUT_SEQ_ON   :=  FALSE;
               END_IF;
               "DC".MOB_FDR_VIB_ON           :=  FALSE;
               "FLT".MOB_FDR_NOT_DCK         :=  FALSE;
               "FLT".MOB_FDR_STP_PARA        :=  FALSE;

               // init magnet
               // -----------
               "DC".MAG_ON := ("AC".SET_MAG_1_CUR > 0.0);                       

               "AC".SET_MAG_1_CUR := "KYA".SET_MAG_1_CUR;
               "AC".SET_MAG_2_CUR := "AC".SET_MAG_1_CUR * "KYA".SET_MAG_RATIO_CUR;

               // init control loops
               // ------------------
               "DC".CTL_DIA_ON       := FALSE;                    // all control loops off
               "DC".CTL_GRW_RTE_ON   := FALSE;
               "DC".CTL_PULL_RTE_ON  := FALSE;
               "DC".CTL_CRUC_ROT_ON  := FALSE;
               "DC".CTL_MLT_LVL_ON   := FALSE;
               "DC".CTL_MLT_1_TMP_ON := FALSE;
               "DC".CTL_MLT_2_TMP_ON := FALSE;
               "DC".CTL_MLT_DRIFT_ON := FALSE;
               "DC".CTL_GAP_ON       := FALSE;

               "DC".CTL_HTR_1_TMP_ON := FALSE;
               "DC".CTL_HTR_2_TMP_ON := FALSE;

               "DC".SET_HTR_1_TMP_ABS := TRUE;            // disable inc functions
               "DC".SET_HTR_2_PWR_ABS := TRUE;  

               "DC".CTL_PRS_ON        := TRUE;

               "DC".CTL_SI_FDR_ON     := FALSE;
               "DC".CTL_DOP_FDR_ON    := FALSE;

               "DV".TRANS_SH_BY_FLAG  := FALSE;
               "DV".START_SH_FLAG     := FALSE;

               "AC".SET_XT_DIA           := 0.0;
               "AC".SET_GRW_RTE          := 0.0;
               "AC".SET_AVG_SPD          := 0.0;
               "AC".SET_AVG_CRUC_ROT     := 0.0;
               "AC".SET_MLT_LVL_LSR      := 0.0;
               "AC".SET_MLT_1_TMP        := "PAR_MAIN".DI_TMP_DIPPING;
               "AC".SET_MLT_2_TMP        := 0.0;
               "AC".SET_HTR_1_TMP_INC    := 0.0;
               "AC".SET_HTR_2_PWR_INC    := 0.0;

               // init measurement system
               // -----------------------
               "DC".CAM_ISP_ON   :=  TRUE;               //inspection on
               "DC".CAM_INIT     :=  FALSE;
               "DC".CAM_MLT      :=  FALSE;
               "DC".CAM_DIP      :=  TRUE;               // switch on dipping mode       
               "DC".CAM_DIA      :=  FALSE;
               "DC".CAM_SEL_1    :=  TRUE;
               "DC".CAM_SEL_2    :=  FALSE;

               "DC".LSR_ON       := FALSE;               // laser off
               "DC".MCC_ON       := FALSE;               // melt contact control off
               "DC".MCC_TST_ON   := FALSE;               // melt contact control test off

               //init setting for camera threshold calculation
               //---------------------------------------------
               "KYA".SET_THR_CAL_FACT              := 1.0;         // default value for threshold ratio factor
             //BM_CAM_THR_CALC_DB.SET_THR_CALC   := 0.0;         // reset value for calculated threshold
               "DV".THR_CALC_ACTIVE                := FALSE;       // set active flag for camera threshold calculation
               "DV".THR_CALC_DISABLED              := FALSE;
             //BM_CAM_THR_CALC_DB.THR_CALC_DONE  := FALSE;


               // init Si feeder system
               // ---------------------
               "DC".SI_FDR_ON    := FALSE;                    // feeder off
               "DC".DOP_FDR_ON   := FALSE;

               "AC".SET_FDR_SI   := 0.0;
               "AC".SET_FDR_DOP  := 0.0;

               // init lamp on control cabinet
               // ----------------------------
               "DV".LMP_OR :=    FALSE; 

               // init timer
               //-----------
               "APC".TI[1]    := 0;

               //init Si charge weight calculation
               //----------------------------------
               "DV".NEW_SI_CRG_WGT_CALC :=  TRUE;

               // calculate all setpoints (step no. from 1st line of sequence table)
               // ----------------------------------------------------------------
               #par_line := 1;
               #par_step := REAL_TO_INT ("PAR_X_VALUES_1".PAR["APC".DIPPING, #par_line]);            
               "AM_PAR_FNC_DI" (act_x_value := #par_step);

               //reset calculation done flag of 2nd crystal length - function call at the end of FB AM_DI
               //----------------------------------------------------------------------------------------
               #xt_lgh_calc_done    := false; 

               //reset calculated weight of grown crystal when dipping is started with remelted previous body
               //--------------------------------------------------------------------------------------------
               IF NOT "APC".CALC_LEN2 THEN
                   "KYA".CALC_WGT_GRW_XT :=  0.0;
                   #prv_calc_wgt_grw_xt :=  0.0;
               END_IF;

               #end_of_step[0]      := true;                            
               #next_step[0]        := 50;

   //-step-50----level--0-------------------------------------------------------------                                                 
   //            DI: gate valve open ?
   //---------------------------------------------------------------------------------                                                 
           50 :                                                     
               IF #next_step[0] = #active_step[0] THEN
                   "APC".OP_MSG := "OP_MSG".WAIT_FOR_AUTO;                                                  
               END_IF;

               IF ("LT".V7_OPEN = TRUE) THEN                    // gate valve open ?
                   // open, enable automatic mode
                   // ---------------------------
                   "DC".MOD_AUT_ENB := TRUE;
                   "FLT".PD_GATE_VALVE_CLOSED := FALSE;
                   #end_of_step[0] := true;
               ELSE
                   // closed, set alarm
                   // -----------------
                   "APC".OP_MSG := "OP_MSG".OPEN_GATE_VALVE;                                                  
                   "DC".MOD_AUT_ENB := FALSE;
                   "FLT".PD_GATE_VALVE_CLOSED := TRUE;
               END_IF;                                    
               #next_step[0] := 100;

   //-step-100---level--0-------------------------------------------------------------                                                 
   //            DI: wait for automatic mode
   //---------------------------------------------------------------------------------                                                 
           100 :                                                     
               IF #next_step[0] = #active_step[0] THEN
                   "APC".OP_MSG := "OP_MSG".WAIT_FOR_AUTO;                                                  
               END_IF;

               IF "APC".AUTOMATIC THEN                    // automatic mode ?
                   #end_of_step[0] := true;                            
               END_IF;                                    
               #next_step[0] := 150;

   //-step-150---level--0-------------------------------------------------------------                                                 
   //            DI: start dipping time
   //---------------------------------------------------------------------------------                                                 
           150 :                                                     
               "APC".ACT_TME_PROC    := 0;                           // start process time
               #end_of_step[0]      := true;                            
               #next_step[0]        := 200;


   //-step-200---level--0-------------------------------------------------------------                                                 
   //            DI: initial power and hold time, move cable and crucible 
   //---------------------------------------------------------------------------------                                                 
           200 :
               IF #next_step[0] = #active_step[0] THEN                  
                   //reset initial temperature and power setpoints
                   //---------------------------------------------
                   "DIS".HTR_1_TMP_SET_PHA_STR   :=  0.0;
                   "DIS".HTR_2_PWR_SET_PHA_STR   :=  0.0;

                   "APC".TI[0] := 0;                     // start step time
               END_IF;

               // fetch actual step time for this step
               // -----------------------------------------------            
               #par_time := REAL_TO_INT ("PAR_TME".PAR["APC".DIPPING, #par_line]);

               // initial heater power
               // --------------------   
               "AC".SET_HTR_1_PWR     := "PAR_MAIN".DI_INI_PWR_1;
               "AC".SET_HTR_2_PWR     := "PAR_MAIN".DI_INI_PWR_2;

               // setpoint magnet
               // ---------------
               "DC".MAG_ON := ("AC".SET_MAG_1_CUR > 0.0);

               "AC".SET_MAG_1_CUR := "AV".SET_MAG_1_CUR;
               "AC".SET_MAG_2_CUR := "AV".SET_MAG_1_CUR * "AV".SET_MAG_RATIO_CUR;


               "APC".OP_MSG := "OP_MSG".DI_1_INIT_TIME;

               // calculate all setpoints for this step
               // -------------------------------------                                      
               "AM_PAR_FNC_DI" (act_x_value := #par_line);

               // setpoint for melt temperature control
               //--------------------------------------
               "AC".SET_MLT_1_TMP    :=    "PAR_MAIN".DI_TMP_DIPPING;
               "AC".SET_HTR_1_TMP    :=    "AV".ACT_HTR_1_TMP; //track heater temperature setpoint with actual value
               (*
               // move crucible
               // -------------
               IF ( (APC.MOVE_CRUC_INTO_DIP_POS = TRUE)
                       AND (KYA.SET_DIP_POS_CR<>0.0)    ) THEN

                   IF (set_cr_pos_old <> KYA.SET_DIP_POS_CR) THEN
                      cruc_in_pos := FALSE;
                   END_IF;

                   DC.CR_LFT_FST := TRUE;
                   AM_DRV_MOVE.AM_CR_DRV_MOVE_DB (   set_pos := KYA.SET_DIP_POS_CR,
                                                     set_spd := CNF.CRUC_LFT_SPEED_FAST,
                                                     act_pos := AV.ACT_CR_POS,
                                                     cnf     := CNF.CNF_CR_POS,
                                                     out_up  := DC.CR_LFT_UP,
                                                     out_dn  := DC.CR_LFT_DN,
                                                     out_spd := AC.SET_CR_SPD,
                                                     done    := cruc_in_pos);

                   IF (cruc_in_pos) THEN
                       set_cr_pos_old := KYA.SET_DIP_POS_CR;
                   END_IF;

               ELSE
                   cruc_in_pos    :=    TRUE;    
               END_IF;
               *)

               // move xtal seed if below upper limit for stabilisation 
               // -----------------------------------------------------
               IF ("AV".ACT_XT_POS > "CNF".DIP_XT_POS AND
                   "AV".ACT_XT_POS > "PAR_MAIN".MCONST_LIM_XTAL_UP) THEN
                     #xtal_in_pos      := FALSE;
                     "DC".XT_LFT_UP     := TRUE;  
                     "DC".XT_LFT_FST    := TRUE;
                     "AC".SET_XT_SPD    := "CNF".DIP_XT_SPD_UP;
               ELSE
                     #xtal_in_pos      := TRUE;
                     "DC".XT_LFT_UP     := FALSE;  
                     "DC".XT_LFT_FST    := FALSE;
                     "AC".SET_XT_SPD    := 0.0;

               END_IF;

               // time till end of this step
               // --------------------------
               IF #par_time >= "APC".TI[0]    THEN
                   "APC".ACT_TME_STE := #par_time - "APC".TI[0];
               ELSE
                   "APC".ACT_TME_STE    :=    0;
               END_IF;

               // end of step 
               // -----------
               IF ("APC".TI[0] > #par_time)       AND
                 //cruc_in_pos    =    true    AND
                   #xtal_in_pos    =    true    THEN
                  #end_of_step[0] := true;
               END_IF;

               #next_step[0] := 250; 

   //-step-250---level--0-------------------------------------------------------------                                                 
   //            DI: set temperature setpoints and wait 
   //---------------------------------------------------------------------------------                                                 
           250 :
               IF #next_step[0] = #active_step[0] THEN   
                    "APC".TI[0] := 0;                     // start step time
               END_IF;

               //absolute mode for heater
               //------------------------
               "DC".SET_HTR_1_TMP_ABS := TRUE;    
               "DC".SET_HTR_2_PWR_ABS := TRUE;
               "AC".SET_HTR_1_TMP     := "AV".ACT_HTR_1_TMP;
               "AC".SET_MLT_1_TMP     := "PAR_MAIN".DI_TMP_DIPPING;

               IF ("APC".TI[0] >= 5) THEN
                     #end_of_step[0] := true;
               END_IF;

               #next_step[0] := 300;

   //-step-300---level--0-------------------------------------------------------------                                                 
   //            DI: switch on temperature control 
   //---------------------------------------------------------------------------------                                                 
           300 :
               IF #next_step[0] = #active_step[0] THEN   
                   "APC".TI[0] := 0;                     // start step time
                   // next line in parameter table
                   // ----------------------------
                   #par_line := #par_line + 1;
                   "APC".OP_MSG := "OP_MSG".DI_2_WAIT_TILL_CTL;
               END_IF;

               // fetch step time of this new line
               // ----------------------------------
               #par_time := REAL_TO_INT ("PAR_TME".PAR["APC".DIPPING, #par_line]);   

               //absolute mode for temp heater 1 mode and power heater 2 mode
               //------------------------------------------------------------
               "DC".SET_HTR_1_TMP_ABS := TRUE;    
               "DC".SET_HTR_2_PWR_ABS := TRUE;

               //set setpoint heater 1 temp = actual filtered temperature
               //--------------------------------------------------------
               "AC".SET_HTR_1_TMP    :=    "AV".ACT_HTR_1_TMP;

               // calculate all setpoints for this step
               // -------------------------------------                                      
               "AM_PAR_FNC_DI" (act_x_value := #par_line);

               // setpoint for melt temperature control
               //--------------------------------------
               "AC".SET_MLT_1_TMP    :=    "PAR_MAIN".DI_TMP_DIPPING;

               // setpoint magnet
               // ---------------
               "DC".MAG_ON := ("AC".SET_MAG_1_CUR > 0.0);

               "AC".SET_MAG_1_CUR := "AV".SET_MAG_1_CUR;
               "AC".SET_MAG_2_CUR := "AV".SET_MAG_1_CUR * "AV".SET_MAG_RATIO_CUR;

               //save crucible position for diping
               //---------------------------------
               "KYA".SET_DIP_POS_CR    :=    "AV".ACT_CR_POS;      

               // time till end of this step
               // --------------------------
               "APC".ACT_TME_STE := #par_time - "APC".TI[0];

               //check deviation from dip temperature, actual melt temperature is used as filtered value
               //------------------------------------
               IF  (("PAR_MAIN".DI_TMP_DIPPING + "PAR_MAIN".DI_TMP_DEV_START) >= "CTL".AVG_MLT_1_TMP) 
                     AND
                   (("PAR_MAIN".DI_TMP_DIPPING - "PAR_MAIN".DI_TMP_DEV_START) <= "CTL".AVG_MLT_1_TMP)
               THEN

               //switch on melt temperature control
               //----------------------------------
                     "DC".CTL_MLT_1_TMP_ON := TRUE;
                     #end_of_step[0] := true;

               //switch on temperature control after max. time
               //---------------------------------------------
               ELSIF ("APC".TI[0] >= #par_time) THEN
                     "DC".CTL_MLT_1_TMP_ON := TRUE;
                     #end_of_step[0] := true;
               END_IF;

               #next_step[0] := 400;

   //-step-400---level--0-------------------------------------------------------------                                                 
   //            DI: melt temperature stabilisation
   //---------------------------------------------------------------------------------                                             
           400 :
                IF #next_step[0] = #active_step[0] THEN  
                   "APC".TI[0] := 0;                     // start step time
                   "APC".OP_MSG := "OP_MSG".DI_3_MELT_TEMP_CTL;
                   //next line in parameter table
                   //----------------------------
                   #par_line := #par_line + 1;

                END_IF;

                // fetch step time of this new line
                // ----------------------------------
                #par_time := REAL_TO_INT ("PAR_TME".PAR["APC".DIPPING, #par_line]);      

                //switch on heater temp control and melt temp control
                //---------------------------------------------------
                "DC".CTL_MLT_1_TMP_ON := TRUE;

                IF ("APC".TI[0] >= 2) THEN 
                   "DC".CTL_HTR_1_TMP_ON := TRUE;
                END_IF;

                "DC".SET_HTR_1_TMP_ABS := FALSE;      //temp heater 1 increment mode     
                "DC".SET_HTR_2_PWR_ABS := FALSE;      //power heater 2 increment mode

                // setpoint magnet
                // ---------------
                "DC".MAG_ON := ("AC".SET_MAG_1_CUR > 0.0);

                "AC".SET_MAG_1_CUR := "AV".SET_MAG_1_CUR;
                "AC".SET_MAG_2_CUR := "AV".SET_MAG_1_CUR * "AV".SET_MAG_RATIO_CUR;


                // calculate all setpoints for this step
                // -------------------------------------                                      
                "AM_PAR_FNC_DI" (act_x_value := #par_line);

                // setpoint for melt temperature control
                //--------------------------------------
                "AC".SET_MLT_1_TMP    :=    "PAR_MAIN".DI_TMP_DIPPING;

                //check if image is ok for dipping after camera is in dipping mode
                //----------------------------------------------------------------
                IF (("APC".ACT_TME_STE <= 0) AND #dip_temp_dev_ok)  THEN
                   IF "DV".CAM_DIP_COMPLETE    THEN
                       "FLT".DI_IMAGE_TO_DARK    :=    TRUE;
                   ELSE
                       "FLT".DI_IMAGE_TO_DARK    :=    FALSE;
                   END_IF; 
                   #dip_image_check := true;
                ELSE
                   #dip_image_check := false;
                END_IF;     

                //check melt contact control function (MCC)
                //----------------------------------------
                IF ("APC".TI[0] < 60) THEN         //check during first minute of step
                   #mcc_error_flag_2:= "DV".DI_MCC_CONTACT;    //melt contact control input error
                END_IF;

                IF ("APC".TI[0] > 60 AND "APC".TI[0] < 120) THEN    //check during second minute of step
                   "DC".MCC_ON := TRUE;                       
                   "DC".MCC_TST_ON := TRUE;
                   #mcc_error_flag_1:= NOT "DV".DI_MCC_CONTACT;    //melt contact control function error
                ELSE    
                   "DC".MCC_TST_ON := FALSE;
                END_IF;

                //check crucible or xtal shaft isolation
                //--------------------------------------
                IF ("APC".TI[0] > 120 AND "APC".TI[0] < 180) THEN    //start test two minutes after step has started 
                   "DC".MCC_ON    :=    TRUE;
                   #mcc_isolation_flag:= "DV".DI_MCC_CONTACT; 
                END_IF;

                //set alarm messages for mcc
                //--------------------------
                IF ("APC".TI[0] > 180) THEN
                   "FLT".DI_ISOLATION_FAULT   := #mcc_isolation_flag;
                   "FLT".DI_MCC_ERROR_1       := #mcc_error_flag_1;
                   "FLT".DI_MCC_ERROR_2       := #mcc_error_flag_2;
                END_IF;

                //check start of min time for constant temperature
                //------------------------------------------------
                IF ((#par_time - "APC".TI[0]) > (REAL_TO_INT("PAR_MAIN".DI_MIN_TME)))      THEN
                    "APC".ACT_TME_STE := #par_time - "APC".TI[0];
                END_IF;

                //reset conditions for min. time for constant temperature
                //-------------------------------------------------------
                IF    #dip_temp_dev_ok    =     FALSE    OR
                      ((#par_time - "APC".TI[0]) > (REAL_TO_INT("PAR_MAIN".DI_MIN_TME)))    THEN    
                      "APC".TI[1]    :=    0;
                END_IF; 

                //min time for constant dip temperature has started
                //-------------------------------------------------
                IF ((#par_time - "APC".TI[0]) <= (REAL_TO_INT("PAR_MAIN".DI_MIN_TME)))    THEN  
                     "APC".ACT_TME_STE := (REAL_TO_INT("PAR_MAIN".DI_MIN_TME) - "APC".TI[1]);           
                END_IF;

                //check actual melt temperature deviation from dip temperature set point
                //---------------------------------------------------------------------- 
                IF (("DIS".SET_MLT_TMP_1 = "AC".SET_MLT_1_TMP)                                     AND 
                   (("PAR_MAIN".DI_TMP_DIPPING + "PAR_MAIN".DI_TMP_DEV_DIP) >= "CTL".AVG_MLT_1_TMP)  AND 
                   (("PAR_MAIN".DI_TMP_DIPPING - "PAR_MAIN".DI_TMP_DEV_DIP) <= "CTL".AVG_MLT_1_TMP)) THEN

                     #dip_temp_dev_ok := TRUE;                 
                //actual melt temperature outside the temperature band
                //---------------------------------------------------- 
                ELSE
                     #dip_temp_dev_ok := FALSE;
                END_IF;

                //check dip condition before switching to next step
                //-------------------------------------------------
                IF ("APC".ACT_TME_STE <= 0) AND #dip_temp_dev_ok AND #dip_image_check THEN
                   #dip_condition_ok    := TRUE;
                ELSE
                   #dip_condition_ok    := FALSE;
                END_IF;

                // end of step ?
                // -------------
                IF #dip_condition_ok    THEN 
                   #end_of_step[0] := true;

                END_IF;

                #next_step[0] := 450;

   //-step-450---level--0-------------------------------------------------------------                                                 
   //            DI: check for mcc and camera errors
   //---------------------------------------------------------------------------------                                                  
           450 :
                //check interlocks for seed lift
                //------------------------------
                IF "FLT".DI_IMAGE_TO_DARK     = FALSE    AND
                   "FLT".DI_ISOLATION_FAULT   = FALSE    AND
                   "FLT".DI_MCC_ERROR_1       = FALSE    AND
                   "FLT".DI_MCC_ERROR_2       = FALSE    THEN
                       #end_of_step[0] := true;
                       #next_step[0] := 500;
                ELSE
                       // stay in this step - operator needs to trigger further actions
                       // -------------------------------------------------------------
                       #next_step[0] := 450;
                END_IF;


   //-step-500---level--0-------------------------------------------------------------                                                 
   //            DI: move down seed (fast speed) with camera detection
   //---------------------------------------------------------------------------------                                                  
           500 :
                IF #next_step[0] = #active_step[0] THEN   
                    "APC".TI[0] := 0;                     // start step time
                    //next line in parameter table
                    //----------------------------
                    #par_line           := #par_line + 1;
                    "APC".OP_MSG         := "OP_MSG".DI_4_SEED_DOWN;
                    "AC".SET_HTR_1_TMP   := "CTL".SET_HTR_1_TMP;
                END_IF;

                // fetch step time of this new line
                // ----------------------------------
                #par_time := REAL_TO_INT ("PAR_TME".PAR["APC".DIPPING, #par_line]);

                //set conditions for this step
                //----------------------------
                "DC".CTL_MLT_1_TMP_ON  := FALSE;
                "DC".CTL_HTR_1_TMP_ON  := TRUE;
                "DC".SET_HTR_1_TMP_ABS := TRUE; 
                "DC".SET_HTR_2_PWR_ABS := FALSE; 
                "DC".MCC_ON            := TRUE;

                // setpoint magnet
                // ---------------
                "DC".MAG_ON := ("AC".SET_MAG_1_CUR > 0.0);

                "AC".SET_MAG_1_CUR := "AV".SET_MAG_1_CUR;
                "AC".SET_MAG_2_CUR := "AV".SET_MAG_1_CUR * "AV".SET_MAG_RATIO_CUR;


                //setpoint xtal speed
                //-------------------
                "AC".SET_XT_SPD := "CNF".XT_LFT_SPEED_FAST;

                // start seed lift down
                //---------------------
                "DC".XT_LFT_DN         := TRUE; 
                "DC".XT_LFT_FST        := TRUE;

                // calculate all setpoints for this step
                // -------------------------------------                                      
                "AM_PAR_FNC_DI" (act_x_value := #par_line);

                // setpoint for melt temperature control
                //--------------------------------------
                "AC".SET_MLT_1_TMP    :=    "PAR_MAIN".DI_TMP_DIPPING;

                // time till end of this step
                // --------------------------
                "APC".ACT_TME_STE := #par_time - "APC".TI[0];

                //fault message if step time is exceeded
                //--------------------------------------
                IF "APC".ACT_TME_STE    <    0    THEN
                    "FLT".DI_TIME_CAM_EXCEEDED    :=    TRUE;
                ELSE
                    "FLT".DI_TIME_CAM_EXCEEDED    :=    FALSE;  
                END_IF;  

                //check camera function and set fault message
                //-------------------------------------------
                IF "DV".DI_MCC_CONTACT    =    TRUE    THEN
                   "FLT".DI_SEED_NOT_CAM_STOPPED    :=    TRUE;
                ELSE
                   "FLT".DI_SEED_NOT_CAM_STOPPED    :=    FALSE;    
                END_IF;

                //end of step
                //stop xtal lift fast speed when camera detects seed 
                //--------------------------------------------------
                IF ("DV".CAM_DIP_COMPLETE OR "DV".DI_MCC_CONTACT OR "DV".ARB_XT_DN_BY_CAM) THEN    
                    "DC".XT_LFT_FST      := FALSE;
                    #end_of_step[0]     := true;
                END_IF;

                #next_step[0] := 600;

   //-step-600---level--0---------------------------------------------------------------                                                 
   //            DI: move down seed (normal speed) into melt with melt contact detection
   //-----------------------------------------------------------------------------------                                               
           600 :            
                IF #next_step[0] = #active_step[0] THEN   
                   "APC".TI[0] := 0;                     // start step time
                   // next line in parameter table
                   // ----------------------------
                   #par_line := #par_line + 1;
                   "APC".OP_MSG := "OP_MSG".DI_5_SEED_INTO_MELT;
                END_IF;

                //reset fault condition from previous step
                //----------------------------------------
                "FLT".DI_TIME_CAM_EXCEEDED    :=    FALSE; 

                // fetch step time of this new line
                // ----------------------------------
                #par_time := REAL_TO_INT ("PAR_TME".PAR["APC".DIPPING, #par_line]);

                //set conditions for this step
                //----------------------------
                "DC".CTL_MLT_1_TMP_ON  := FALSE;
                "DC".CTL_HTR_1_TMP_ON  := TRUE;
                "DC".SET_HTR_1_TMP_ABS := TRUE;   
                "DC".SET_HTR_2_PWR_ABS := FALSE;         
                "DC".XT_LFT_DN         := TRUE; 
                "DC".XT_LFT_FST        := FALSE;
                "DC".MCC_ON            := TRUE;

                "AC".SET_XT_SPD        :=    "CNF".XT_LFT_SPEED_NORM;

                // setpoint magnet
                // ---------------
                "DC".MAG_ON := ("AC".SET_MAG_1_CUR > 0.0);

                "AC".SET_MAG_1_CUR := "AV".SET_MAG_1_CUR;
                "AC".SET_MAG_2_CUR := "AV".SET_MAG_1_CUR * "AV".SET_MAG_RATIO_CUR;

                // calculate all setpoints for this step
                // -------------------------------------                                      
                "AM_PAR_FNC_DI" (act_x_value := #par_line);

                // setpoint for melt temperature control
                //--------------------------------------
                "AC".SET_MLT_1_TMP    :=    "PAR_MAIN".DI_TMP_DIPPING;

                // time till end of this step
                // --------------------------
                "APC".ACT_TME_STE := #par_time - "APC".TI[0];

                //fault message if step time is exceeded
                //--------------------------------------
                IF ("APC".ACT_TME_STE < 0)    THEN                
                    "FLT".DI_TIME_MELT_EXCEEDED    :=    TRUE; 
                ELSE
                    "FLT".DI_TIME_MELT_EXCEEDED    :=    FALSE; 
                END_IF;

                //end of step
                //stop xtal lift norm speed with delay time when seed dips into melt 
                //------------------------------------------------------------------
                IF "DV".DI_MCC_CONTACT = FALSE    THEN
                   "APC".TI[1]    :=    0;
                END_IF;

                IF ("DV".DI_MCC_CONTACT AND "APC".TI[1] > 45)    = TRUE    THEN    
                    "DC".XT_LFT_DN         := FALSE;
                    #end_of_step[0]       := true;
                END_IF;

                #next_step[0] := 700;

   //-step-700---level--0-------------------------------------------------------------                                                 
   //            DI: WAIT TIME 1
   //---------------------------------------------------------------------------------                                                 
           700 :
                IF #next_step[0] = #active_step[0] THEN   
                   "APC".TI[0] := 0;                     // start step time
                   // next line in parameter table
                   // ----------------------------
                   #par_line := #par_line + 1;
                   "APC".OP_MSG := "OP_MSG".DI_6_WAIT_TIME1;
                END_IF;

                //reset fault condition from previous step
                //----------------------------------------
                "FLT".DI_TIME_MELT_EXCEEDED    :=    FALSE; 

                // fetch step time of this new line
                // ----------------------------------
                #par_time := REAL_TO_INT ("PAR_TME".PAR["APC".DIPPING, #par_line]);

                //set conditions for this step
                //----------------------------
                "DC".CTL_MLT_1_TMP_ON  := FALSE;
                "DC".CTL_HTR_1_TMP_ON  := TRUE;
                "DC".SET_HTR_1_TMP_ABS := TRUE; 
                "DC".SET_HTR_2_PWR_ABS := FALSE;           
                "DC".XT_LFT_DN         := FALSE; 
                "DC".XT_LFT_FST        := FALSE;
                "DC".MCC_ON            := FALSE;

                //reset speed setpoint
                //--------------------
                "AC".SET_XT_SPD        := 0.0;

                // setpoint magnet
                // ---------------
                "DC".MAG_ON := ("AC".SET_MAG_1_CUR > 0.0);

                "AC".SET_MAG_1_CUR := "AV".SET_MAG_1_CUR;
                "AC".SET_MAG_2_CUR := "AV".SET_MAG_1_CUR * "AV".SET_MAG_RATIO_CUR;

                // calculate all setpoints for this step
                // -------------------------------------                                      
                "AM_PAR_FNC_DI" (act_x_value := #par_line);

                // setpoint for melt temperature control
                //--------------------------------------
                "AC".SET_MLT_1_TMP    :=    "PAR_MAIN".DI_TMP_DIPPING;

                // time till end of this step
                // --------------------------
                "APC".ACT_TME_STE := #par_time - "APC".TI[0];

                //end of step
                //-----------
                IF ("APC".TI[0] > #par_time) THEN
                  #end_of_step[0] := true;
                END_IF;

                #next_step[0] := 800;

   //-step-800---level--0-------------------------------------------------------------                                                 
   //            DI: WAIT TIME 2
   //---------------------------------------------------------------------------------                                               
           800 :
                IF #next_step[0] = #active_step[0] THEN   
                   "APC".TI[0] := 0;                     // start step time
                   // next line in parameter table
                   // ----------------------------
                   #par_line        := #par_line + 1;
                   "APC".OP_MSG      := "OP_MSG".DI_7_WAIT_TIME2;

                END_IF;

                // fetch step time of this new line
                // ----------------------------------
                #par_time := REAL_TO_INT ("PAR_TME".PAR["APC".DIPPING, #par_line]);

                //set conditions for this step
                //----------------------------
                "DC".CTL_MLT_1_TMP_ON  := FALSE;
                "DC".CTL_HTR_1_TMP_ON  := TRUE;
                "DC".SET_HTR_1_TMP_ABS := TRUE; 
                "DC".SET_HTR_2_PWR_ABS := FALSE;           
                "DC".XT_LFT_DN         := FALSE; 
                "DC".XT_LFT_FST        := FALSE;
                "DC".MCC_ON            := FALSE;

                //temperature setpoint
                //--------------------
                #htr_1_tmp_before_gap     := "CTL".SET_HTR_1_TMP;    //save heater 1 temp before gap

                // setpoint magnet
                // ---------------
                "DC".MAG_ON := ("AC".SET_MAG_1_CUR > 0.0);

                "AC".SET_MAG_1_CUR := "AV".SET_MAG_1_CUR;
                "AC".SET_MAG_2_CUR := "AV".SET_MAG_1_CUR * "AV".SET_MAG_RATIO_CUR;

                // calculate all setpoints for this step
                // -------------------------------------                                      
                "AM_PAR_FNC_DI" (act_x_value := #par_line);

                // setpoint for melt temperature control
                //--------------------------------------
                "AC".SET_MLT_1_TMP    :=    "PAR_MAIN".DI_TMP_DIPPING;

                // time till end of this step
                // --------------------------
                "APC".ACT_TME_STE := #par_time - "APC".TI[0];

                //end of step
                //-----------
                IF ("APC".TI[0] > #par_time) THEN
                  #end_of_step[0] := true;
                END_IF;

                #next_step[0] := 900;

   //-step-900---level--0-------------------------------------------------------------                                                 
   //            DI: TEMPERATURE GAP
   //---------------------------------------------------------------------------------                                 
           900 :
                IF #next_step[0] = #active_step[0] THEN   
                   "APC".TI[0] := 0;                     // start step time
                   // next line in parameter table
                   // ----------------------------
                   #par_line := #par_line + 1;
                   "APC".OP_MSG := "OP_MSG".DI_8_TEMP_GAP;
                END_IF;

                //fetch step time of this new line
                //--------------------------------
                #par_time := REAL_TO_INT ("PAR_TME".PAR["APC".DIPPING, #par_line]);

                //set conditions for this step
                //----------------------------
                "DC".CTL_MLT_1_TMP_ON  := FALSE;
                "DC".CTL_HTR_1_TMP_ON  := TRUE;
                "DC".SET_HTR_1_TMP_ABS := TRUE;
                "DC".SET_HTR_2_PWR_ABS := FALSE;           
                "DC".XT_LFT_DN         := FALSE; 
                "DC".XT_LFT_FST        := FALSE;
                "DC".MCC_ON            := FALSE;

                //setpoint calculation temperature gap
                //------------------------------------
                "AC".SET_HTR_1_TMP     :=    #htr_1_tmp_before_gap - "PAR_MAIN".DI_TMP_GAP_HTR_1 - "PAR_MAIN".DI_TMP_DEC_HTR_1;

                // setpoint magnet
                // ---------------
                "DC".MAG_ON := ("AC".SET_MAG_1_CUR > 0.0);

                "AC".SET_MAG_1_CUR := "AV".SET_MAG_1_CUR;
                "AC".SET_MAG_2_CUR := "AV".SET_MAG_1_CUR * "AV".SET_MAG_RATIO_CUR;

                // calculate all setpoints for this step
                // -------------------------------------                                      
                "AM_PAR_FNC_DI" (act_x_value := #par_line);

